(*			
	EVERDE sp. z o.o.
	Rafał Osajda		22.01.2025		TC 4026.13		wer. 0.0.0.1
	B_Baza dla czujników binarnych 	
*)
INTERFACE ITF_Sensor EXTENDS ITF_BaseComponent

(*			
	EVERDE sp. z o.o.
	Rafał Osajda		05.02.2025		TC 4026.13		wer. 0.0.0.1
	Zwraca aktualny stan czujnika
*)
METHOD IsActive : BOOL
END_METHOD

END_INTERFACE

(* stored: Version 1.1.0.1
   Itf ITF_Sensor: Id {b8976a09-76d2-42f1-b965-e778286c6c94}
   Method IsActive: Id {ddb24e15-3ec4-4882-89dc-a61bbd27327b} *)
